# EPICS substitutions: pmacUtilApp/Db/pmacGPOutput.substitutions
file "db/pmacGPOutput.db"
{
pattern
{ SYS,			DEV,		NUM, 		VAR		}
{ "XF:X17A",	"{MC:1}"	1,			"M32"	}
{ "XF:X17A",	"{MC:1}"	2,			"M33"	}
{ "XF:X17A",	"{MC:1}"	3,			"M34"	}
{ "XF:X17A",	"{MC:1}"	4,			"M35"	}
{ "XF:X17A",	"{MC:1}"	5,			"M36"	}
{ "XF:X17A",	"{MC:1}"	6,			"M37"	}
{ "XF:X17A",	"{MC:1}"	7,			"M38"	}
{ "XF:X17A",	"{MC:1}"	8,			"M39"	}
}
